FUNCTION roundToTwoDecimalPlaces:LREAL
VAR_INPUT
	val:LREAL;
END_VAR
VAR_OUTPUT
	rval:LREAL;
END_VAR
VAR
	value:LREAL;
END_VAR

  value := LREAL_TO_DINT(val * 100 + 0.5);
  rval:= value/100;
  roundToTwoDecimalPlaces:=rval;

END_FUNCTION

(* stored: Version 1.1.0.1, ProductVersion 3.1.4024.12
   POU roundToTwoDecimalPlaces: Id {e7da07fe-d52a-4acf-9867-882ee4692ba3}, SpecialFunc None *)
